// TIA Portal V17 export
// export: Created 2025-06-25T13:13:31.8126982Z, ExportSetting WithDefaults, DisplayName Totally Integrated Automation Portal, DisplayVersion V17 Update 8, DisplayName TIA Portal Openness, DisplayVersion V17 Update 8, DisplayName TIA Portal Version Control Interface, DisplayVersion V17, DisplayName STEP 7 Professional, DisplayVersion V17 Update 8, DisplayName STEP 7 Safety, DisplayVersion V17 Update 6, DisplayName WinCC Advanced, DisplayVersion V17 Update 8
TYPE "stOilSeparator"
// stored: IsFailsafeCompliant false
   STRUCT
      Stage1 : "stOnOffRegulator2";
      Stage2 { S7_SetPoint := 'True'} : "stOnOffRegulator2";
   END_STRUCT;
END_TYPE
